(* PLC project RedLine3, Beckhoff Automation GmbH TwinCAT PLC Control 3.5.13.21 *)
(* stored: creationDateTime 2022-07-30T14:47:54.2878237, modificationDateTime 2022-07-30T14:47:54.2918246 *)

PROGRAM MAIN
VAR

inc1 : DINT := 0;
	
END_VAR

            //0 to 37 map to blocks 1-38
//39 to 44 map to blocks 72-76,yard
FOR inc1 := 0 TO 44 DO

	GVL.mOutOccupancies[inc1] := GVL.mInOccupancies[inc1];
	GVL.mOutSpeeds[inc1] := GVL.mInSpeeds[inc1];
	GVL.mOutAuthorities[inc1] := GVL.mInAuthorities[inc1];
	GVL.mOutMaintenance[inc1] := GVL.mInMaintenance[inc1];
	
END_FOR

FOR inc1 := 0 TO 44 DO

	GVL.mOutRoute[inc1] := GVL.mInRoute[inc1];
	
END_FOR

inc1 := 0;

//This starts the main track logic section

//0 to 37 map to blocks 1-38
//39 to 44 map to 72-76,yard
//Switch Logic
IF GVL.mInMaintenance[8] = 1 THEN
    GVL.mOutSwitch[8] := GVL.mInSwitch[8];
ELSE
    IF GVL.mInOccupancies[43] = 0 THEN
    	GVL.mOutSwitch[8] := 76;
    ELSE
		GVL.mOutSwitch[8] := 9;
	END_IF
END_IF

//0 to 37 map to blocks 1-38
//39 to 44 map to 72-76,yard
IF GVL.mInMaintenance[15] = 1 THEN
    GVL.mOutSwitch[15] := GVL.mInSwitch[15];
ELSE
    IF GVL.mInOccupancies[14] = 0 THEN
    FOR inc1 := 16 TO 26 DO 
        IF GVL.mInOccupancies[inc1] = 0 THEN
            GVL.mOutSwitch[15] := 1;
            Exit;
        ELSE 
            GVL.mOutSwitch[15] := 14;
        END_IF
    END_FOR
	END_IF
END_IF

//0 to 37 map to blocks 1-38
//39 to 44 map to 72-76,yard
IF GVL.mInMaintenance[26] = 1 THEN
    GVL.mOutSwitch[26] := GVL.mInSwitch[26];
ELSE
    IF GVL.mInOccupancies[43] = 0 THEN
    FOR inc1 := 16 TO 26 DO 
        IF GVL.mInOccupancies[inc1] = 0 THEN
            GVL.mOutSwitch[26] := 27;
            Exit;
        ELSE 
            GVL.mOutSwitch[26] := 75;
        END_IF
    END_FOR
	END_IF
END_IF

//0 to 37 map to blocks 1-38
//39 to 44 map to 72-76,yard
IF GVL.mInMaintenance[32] = 1 THEN
    GVL.mOutSwitch[32] := GVL.mInSwitch[32];
ELSE
    IF GVL.mInOccupancies[31] = 0 THEN
    FOR inc1 := 32 TO 37 DO 
        IF GVL.mInOccupancies[inc1] = 0 THEN
            GVL.mOutSwitch[32] := 71;
            Exit;
        ELSE 
            GVL.mOutSwitch[32] := 31;
        END_IF
    END_FOR
	END_IF
END_IF

          
END_PROGRAM
